(* PLC project  *)

PROGRAM SequenceXml
  VAR
    Ready : BOOL;
    Done : BOOL;
    Count : INT;
  END_VAR

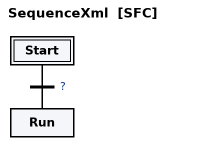
INITIAL_STEP Start:
END_STEP
TRANSITION FROM Start TO Run
  := ?;
END_TRANSITION
STEP Run:
END_STEP
END_PROGRAM
